ABB RobotStudio station: Proyecto_20220130-232737.rsstn

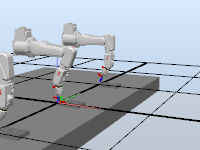
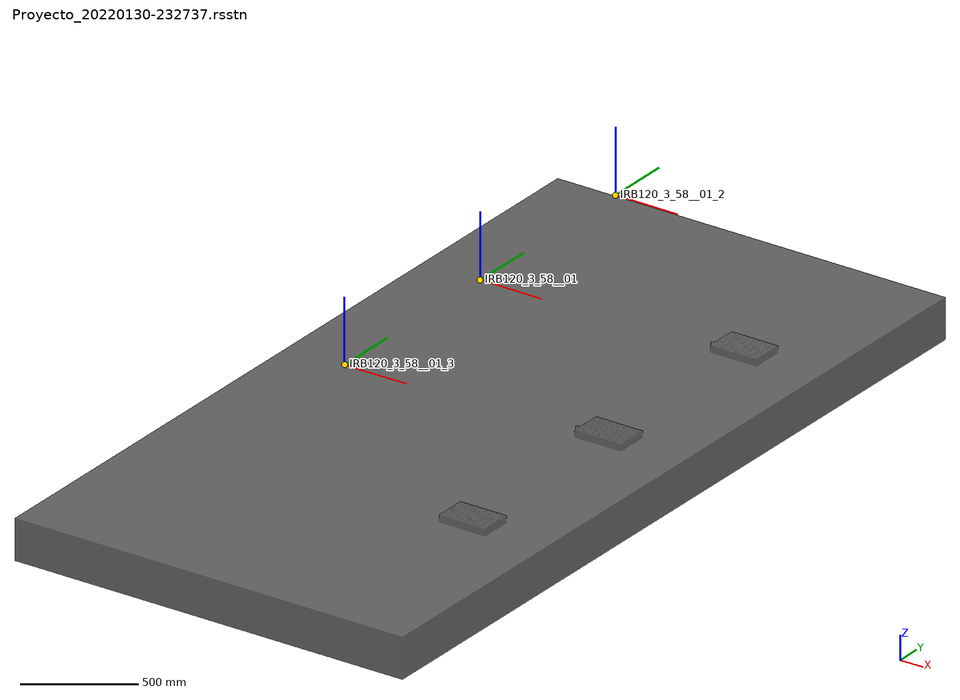
[picture v1: parts stored in the station drawn from their meshes, with robot base, taught points and paths (robot models come from the ABB library and are not in the file)]
Station Proyecto (saved by RobotStudio 21.4.9700.0)
Controller Controlador1, task T_ROB3: task frame (RAPID world) sits at (0, 0, 800) mm, rotated rx 0 ry 90 rz 0 deg in the station
Controller Controlador1, task T_ROB2: task frame (RAPID world) sits at (0, 0, 800) mm, rotated rx 0 ry 90 rz 0 deg in the station
Controller Controlador1, task T_ROB1: task frame (RAPID world) sits at (0, 0, 800) mm, rotated rx 0 ry 90 rz 0 deg in the station
Controller Controlador1
  mechanical unit ROB_1: IRB120_3_58__01, 6 joints, base frame (0, 0, 0) mm
  mechanical unit ROB_2: IRB120_3_58__01_2, 6 joints, base frame (0, 1000, 0) mm
  mechanical unit ROB_3: IRB120_3_58__01_3, 6 joints, base frame (0, -1000, 0) mm
Layout (positions relative to the parent item):
  - IRB120_3_58__01 [mechanism, from Robots\IRB120_3_58_G_01.rslib] at (0, 0, 800) mm, rotated rx 0 ry 90 rz 0 deg; joint values [0, 0.087, 0.3322, 0, -0.4192, 0] (rad or m)
  - IRB120_3_58__01_2 [mechanism, from Robots\IRB120_3_58_G_01.rslib] at (0, 1000, 800) mm, rotated rx 0 ry 90 rz 0 deg; joint values [0, 0, 0, 0, 0.5236, 0] (rad or m)
  - IRB120_3_58__01_3 [mechanism, from Robots\IRB120_3_58_G_01.rslib] at (0, -1000, 800) mm, rotated rx 0 ry 90 rz 0 deg; joint values [0, 0, 0, 0, 0.5236, 0] (rad or m)
  - Mesa [part], size 2000 x 4000 x 200 mm
  - Soporte [part] at (500, 0, 251) mm, size 240 x 160 x 36 mm
  - Frasco [part] at (500, 0, 251) mm, size 15 x 15 x 53 mm
  - Smart_Gripper_Servo_Fingers [mechanism, from Tools\ABB_Smart_Gripper_Servo_Fingers.rslib] at (500, 0, 400.2) mm, rotated rx 180 ry 0 rz 180 deg; joint values [0] (rad or m)
  - Smart_Gripper_Servo_Fingers_2 [mechanism, from Tools\ABB_Smart_Gripper_Servo_Fingers.rslib] at (594, 1000, 435.65) mm, rotated rx 180 ry -30 rz 180 deg; joint values [0] (rad or m)
  - Smart_Gripper_Servo_Fingers_3 [mechanism, from Tools\ABB_Smart_Gripper_Servo_Fingers.rslib] at (594, -1000, 435.65) mm, rotated rx 180 ry -30 rz 180 deg; joint values [0] (rad or m)
  - Soporte Tapas [part] at (500, 1000, 200) mm, size 240 x 160 x 36 mm
  - Soporte_2 [part] at (500, -1000, 251) mm, size 240 x 160 x 36 mm
  - Tapa [part] at (500, 1000, 249) mm, rotated rx 180 ry 0 rz 0 deg, size 15 x 15 x 23 mm
  - UCS [frame] at (492, -8, 236) mm
Attachment: Smart_Gripper_Servo_Fingers is attached to IRB120_3_58__01 / Link6
Attachment: Smart_Gripper_Servo_Fingers_2 is attached to IRB120_3_58__01_2 / Link6
Attachment: Smart_Gripper_Servo_Fingers_3 is attached to IRB120_3_58__01_3 / Link6
Targets, tools, work objects and paths stored in the station, written as RAPID:
! task T_ROB1
MODULE CalibData
  PERS tooldata Servo:=[TRUE,[[0,0,114.2],[1,0,0,0]],[0.215,[8.7,12.3,49.2],[1,0,0,0],0.00021,0.00024,0.00009]];
  TASK PERS wobjdata Workobject_2:=[FALSE,TRUE,"",[[564,-8,492],[0.707106781,0,-0.707106781,0]],[[8,8,15],[1,0,0,0]]];
ENDMODULE

! task T_ROB1
MODULE Module1
  PROC Path_10()
    MoveL Target_30,v100,z50,Servo\WObj:=Workobject_2;
  ENDPROC
ENDMODULE

! task T_ROB2
MODULE CalibData
  PERS tooldata Servo:=[TRUE,[[0,0,114.2],[1,0,0,0]],[0.215,[8.7,12.3,49.2],[1,0,0,0],0.00021,0.00024,0.00009]];
ENDMODULE

! task T_ROB3
MODULE CalibData
  PERS tooldata Servo:=[TRUE,[[0,0,114.2],[1,0,0,0]],[0.215,[8.7,12.3,49.2],[1,0,0,0],0.00021,0.00024,0.00009]];
ENDMODULE

